FUNCTION_BLOCK FB_MessageRecording
VAR_INPUT
END_VAR
VAR_OUTPUT
END_VAR
VAR
END_VAR

IF GVL_Global.stGamePlay.sMessageType.bMessageToBeRecorded THEN
	IF GVL_Global.stGamePlay.sMessageType.bErrorMessage THEN
		;
	ELSIF GVL_Global.stGamePlay.sMessageType.bFeedbackMessage THEN
		;
	ELSIF GVL_Global.stGamePlay.sMessageType.bInstructionMessage THEN
		;
	END_IF
END_IF

END_FUNCTION_BLOCK

(* stored: Version 1.1.0.1, ProductVersion 3.1.4024.10
   POU FB_MessageRecording: Id {683ed490-e03e-4e98-9147-912713b63a7b}, SpecialFunc None *)
